FUNCTION mat3Vec3 : vec3d
VAR_IN_OUT CONSTANT
	i_mat :Mat3d;
	i_vec :Vec3d;
END_VAR
VAR
	i,j : INT ;
END_VAR

FOR i:=1 TO 3 DO
	mat3Vec3[i]:=0.0;
	FOR j:=1 TO 3 DO
		mat3Vec3[i]:=mat3Vec3[i]+i_mat[i,j]*i_vec[j];
	END_FOR
END_FOR

END_FUNCTION

(* stored: Version 1.1.0.1, ProductVersion 3.1.4024.12
   POU mat3Vec3: Id {8370fc65-efef-4038-9c46-489d211f783c}, SpecialFunc None *)
